FUNCTION F_GetSubSystemExternErrorData : ST_ErrorDataSet
(**************************************************************************************
 * 	Application		:	BoxControl Framework
 *	Revision		:	$Revision: 404529 $
 *	Revision date	:	$Date: 2018-04-23 08:21:38 +0200 (Mo., 23 Apr 2018) $
 *	Last changed by	:	$Author: b7bolm $
 *	URL				:	$URL: http://almscdc.swisslog.com/repo/SWPD/Development/BoxControlFramework/20_Release/trunk/01_Software/BCF/BCF/JumpStart/20_Product/10_App/15_Subsystem/10_Lib/10_Conv/10_Functions/F_GetSubSystemExternErrorData.TcPOU $
 *
 *	Purpose			:	Return subsystem error data
 *
 * ------------------------------------------------------------------------------------
 *	Copyright Swisslog [IP AG], Switzerland. All rights reserved.
 * 
 * ------------------------------------------------------------------------------------
 *	
 * 	Revision History: 
 *
 * 	VERSION			DATE			INITIALS			DESCRIPTION
 *	0.1				01.01.2001		swl					Example
 *
 **************************************************************************************)


// Check reference is valid
IF __ISVALIDREF(Subsystemregistry.rSubsystemData) THEN
	// Return error data
	F_GetSubSystemExternErrorData :=Subsystemregistry.rSubsystemData.ErrorData.ExternalError;
END_IF

END_FUNCTION

(* stored: Version 1.1.0.1, ProductVersion 3.1.4022.12
   POU F_GetSubSystemExternErrorData: Id {e86b6a0b-e5b4-46c9-95c3-9ac7e333d3a9}, SpecialFunc None *)
